// Mitsubishi GX Works2 project: SmartFarmDXyzSandbox   PLC: FX3U/FX3UC

PROGRAM MAIN
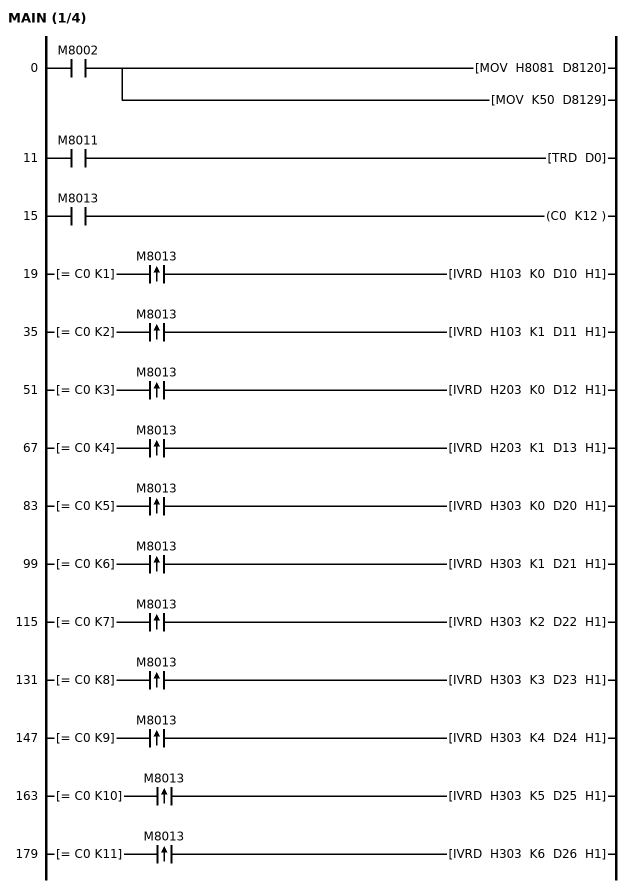
0     LD      M8002
      MOV     H8081 D8120
      MOV     K50 D8129
11    LD      M8011
      TRD     D0
15    LD      M8013
      OUT     C0 K12
19    LD=     C0 K1
      ANDP    M8013
      IVRD    H103 K0 D10 H1
35    LD=     C0 K2
      ANDP    M8013
      IVRD    H103 K1 D11 H1
51    LD=     C0 K3
      ANDP    M8013
      IVRD    H203 K0 D12 H1
67    LD=     C0 K4
      ANDP    M8013
      IVRD    H203 K1 D13 H1
83    LD=     C0 K5
      ANDP    M8013
      IVRD    H303 K0 D20 H1
99    LD=     C0 K6
      ANDP    M8013
      IVRD    H303 K1 D21 H1
115   LD=     C0 K7
      ANDP    M8013
      IVRD    H303 K2 D22 H1
131   LD=     C0 K8
      ANDP    M8013
      IVRD    H303 K3 D23 H1
147   LD=     C0 K9
      ANDP    M8013
      IVRD    H303 K4 D24 H1
163   LD=     C0 K10
      ANDP    M8013
      IVRD    H303 K5 D25 H1
179   LD=     C0 K11
      ANDP    M8013
      IVRD    H303 K6 D26 H1
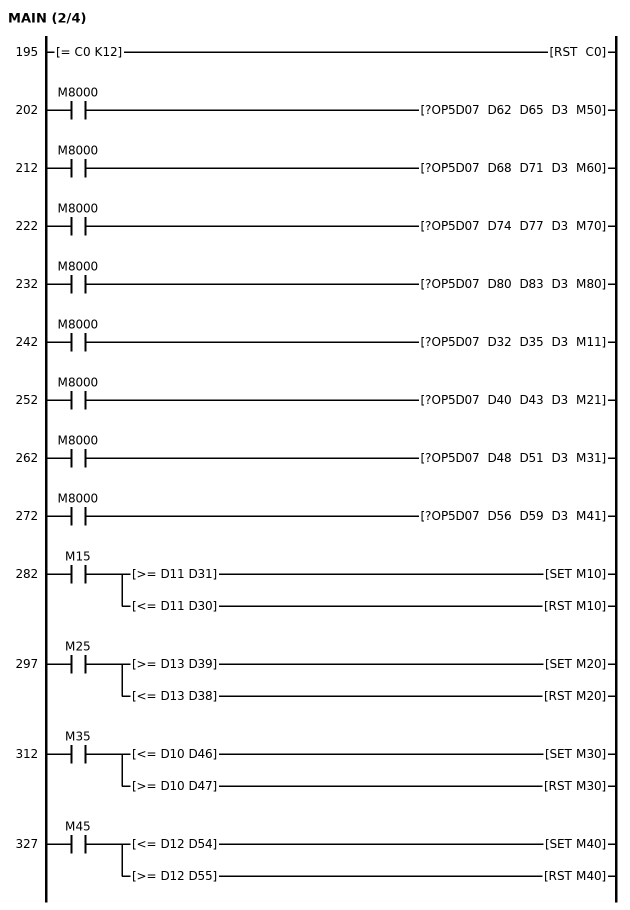
195   LD=     C0 K12
      RST     C0
202   LD      M8000
      ?OP5D07 D62 D65 D3 M50
212   LD      M8000
      ?OP5D07 D68 D71 D3 M60
222   LD      M8000
      ?OP5D07 D74 D77 D3 M70
232   LD      M8000
      ?OP5D07 D80 D83 D3 M80
242   LD      M8000
      ?OP5D07 D32 D35 D3 M11
252   LD      M8000
      ?OP5D07 D40 D43 D3 M21
262   LD      M8000
      ?OP5D07 D48 D51 D3 M31
272   LD      M8000
      ?OP5D07 D56 D59 D3 M41
282   LD      M15
      MPS
      AND>=   D11 D31
      SET     M10
      MPP
      AND<=   D11 D30
      RST     M10
297   LD      M25
      MPS
      AND>=   D13 D39
      SET     M20
      MPP
      AND<=   D13 D38
      RST     M20
312   LD      M35
      MPS
      AND<=   D10 D46
      SET     M30
      MPP
      AND>=   D10 D47
      RST     M30
327   LD      M45
      MPS
      AND<=   D12 D54
      SET     M40
      MPP
      AND>=   D12 D55
      RST     M40
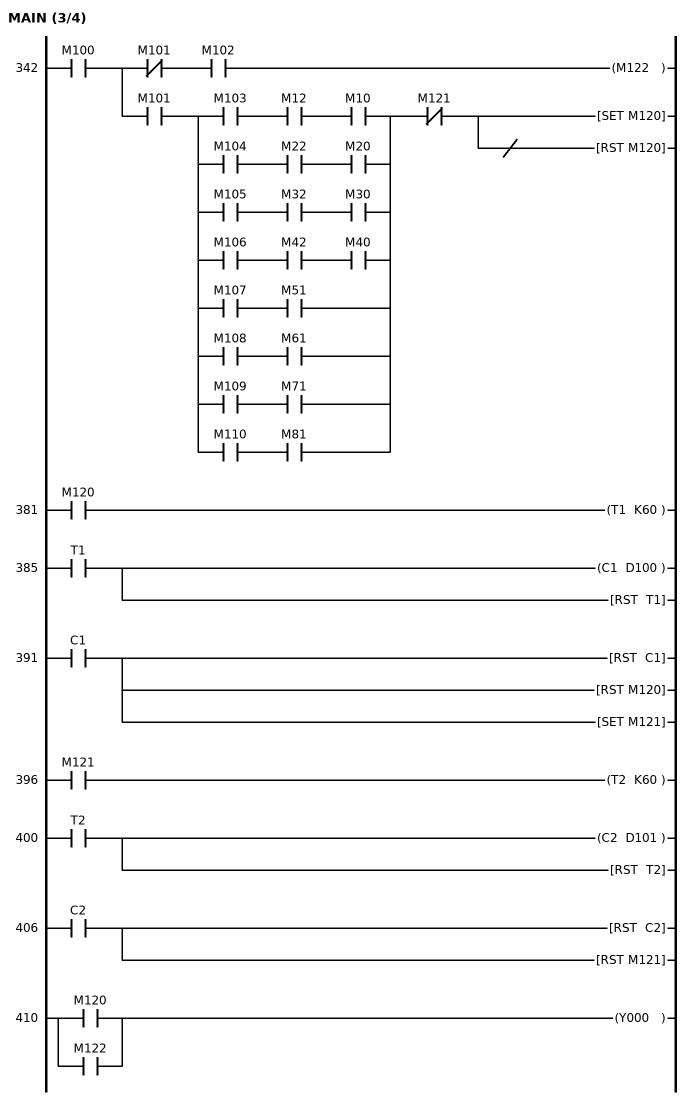
342   LD      M100
      MPS
      ANI     M101
      AND     M102
      OUT     M122
      MPP
      AND     M101
      LD      M103
      AND     M12
      AND     M10
      LD      M104
      AND     M22
      AND     M20
      ORB
      LD      M105
      AND     M32
      AND     M30
      ORB
      LD      M106
      AND     M42
      AND     M40
      ORB
      LD      M107
      AND     M51
      ORB
      LD      M108
      AND     M61
      ORB
      LD      M109
      AND     M71
      ORB
      LD      M110
      AND     M81
      ORB
      ANB
      ANI     M121
      SET     M120
      INV
      RST     M120
381   LD      M120
      OUT     T1 K60
385   LD      T1
      OUT     C1 D100
      RST     T1
391   LD      C1
      RST     C1
      RST     M120
      SET     M121
396   LD      M121
      OUT     T2 K60
400   LD      T2
      OUT     C2 D101
      RST     T2
406   LD      C2
      RST     C2
      RST     M121
410   LD      M120
      OR      M122
      OUT     Y000
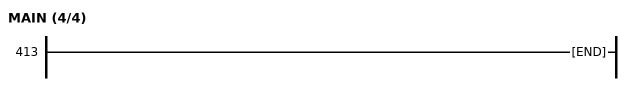
413   END
END_PROGRAM
